FUNCTION cross : Vec3d
VAR_IN_OUT CONSTANT
	a, b :Vec3d;
END_VAR
VAR
END_VAR

cross[1]:=a[2]*b[3]-a[3]*b[2];
cross[2]:=a[3]*b[1]-a[1]*b[3];
cross[3]:=a[1]*b[2]-a[2]*b[1];

END_FUNCTION

(* stored: Version 1.1.0.1, ProductVersion 3.1.4024.12
   POU cross: Id {c93e3312-b801-4db9-af16-39772db794e7}, SpecialFunc None *)
